FUNCTION_BLOCK FB_JanitzaSensor EXTENDS FB_Sensor
VAR_INPUT
END_VAR
VAR_OUTPUT
	fPower : REAL; //measured power in watt
END_VAR
VAR
	//I/O-Links
	power_IN AT %I* : REAL;
	
END_VAR

METHOD GetState_AI : BOOL
VAR_INPUT
END_VAR
fPower := power_IN;

//sensor state
sensorState.fValue := fPower;
sensorState.sUnit := 'Watt';
END_METHOD

END_FUNCTION_BLOCK

(* stored: Version 1.1.0.1, ProductVersion 3.1.4024.6
   POU FB_JanitzaSensor: Id {8fa913e5-ea73-49cb-856e-4271c00e3919}, SpecialFunc None
   Method GetState_AI: Id {bfc089cb-51c5-4333-ac4c-1dfe775f2223} *)
